FUNCTION_BLOCK FB_BacklashCompensationNC_TestDouble IMPLEMENTS I_BacklashCompensation
VAR
END_VAR

{warning 'Add property implementation'}
PROPERTY Aborted : BOOL
GET
END_GET
END_PROPERTY

{warning 'Add property implementation'}
PROPERTY ActCompensation : LREAL
GET
END_GET
END_PROPERTY

{warning 'Add property implementation'}
PROPERTY Active : BOOL
GET
END_GET
END_PROPERTY

{warning 'Add method implementation '}
(*
    Handle positive/negative backlash compensation
    User needs to set the direction of backlash from the sign of the compensation value
    Backlash compensation is disabled during referencing (homing).
    When direction is positive/negative, further movement in the negative/positive direction not compensated
    further movement in the negative/positive direction will be compensated
*)
METHOD BacklashCompensation
VAR_INPUT
    Activate	: BOOL;
    DisableMode	: E_DISABLEMODE := .E_DISABLEMODE.DisableModeHold;
END_VAR
END_METHOD

{warning 'Add property implementation'}
PROPERTY Busy : BOOL
GET
END_GET
END_PROPERTY

{warning 'Add property implementation'}
PROPERTY Done : BOOL
GET
END_GET
END_PROPERTY

{warning 'Add property implementation'}
PROPERTY Error : BOOL
GET
END_GET
END_PROPERTY

{warning 'Add property implementation'}
PROPERTY ErrorID : UDINT
GET
END_GET
END_PROPERTY

{warning 'Add property implementation'}
PROPERTY Message : T_MAXSTRING
GET
END_GET
END_PROPERTY

END_FUNCTION_BLOCK

(* stored: Version 1.1.0.1
   POU FB_BacklashCompensationNC_TestDouble: Id {c8ccd65b-c409-4be0-a30d-cd79c23753d7}, SpecialFunc None
   Property Aborted: Id {babb711a-142f-4c3f-b217-2d95daf21339}
   Get Get: Id {fa604682-deb3-4467-867f-16b2b61c8044}
   Property ActCompensation: Id {24a13000-c259-4876-8f45-c763522d1562}
   Get Get: Id {3671a0ac-cd0b-430f-8ff6-a4fc7ae557dc}
   Property Active: Id {7c066d8d-a8ce-4565-be37-8b7a22588e80}
   Get Get: Id {166665cc-5fed-4c2f-b84a-e7fe59ef0640}
   Method BacklashCompensation: Id {82ce2826-5294-43a2-87fa-a5c006c9feed}
   Property Busy: Id {92ed6e4a-bb6b-4b21-9c22-86522d2aa452}
   Get Get: Id {6936a108-332f-4fed-9b26-8a4d0fde3a28}
   Property Done: Id {a0a34c4a-c99f-4419-9f9f-4d50d2dd02e2}
   Get Get: Id {62ee98f4-ddc7-4c2c-8de5-097bc578d461}
   Property Error: Id {94aa4214-8aad-44ef-968d-20b08e505fb8}
   Get Get: Id {b7f678bc-91bd-4726-9d6c-b6f27975b65c}
   Property ErrorID: Id {50a0126f-1bbc-483e-b6fa-49004da3b45e}
   Get Get: Id {be7639ad-a2b1-4f76-89d0-d51327e167a0}
   Property Message: Id {09310ee4-2e52-4c89-aee3-8d8a5df71d38}
   Get Get: Id {d3035c2f-1387-4860-acc1-41b5a65fdc56} *)
